{attribute 'qualified_only'}
{attribute 'strict'}
TYPE ERetargetType :
(
	not_retargeted := 0,
	primitive_target := 1,
	sequence_target := 2
);
END_TYPE

(* stored: Version 1.1.0.1, ProductVersion 3.1.4024.9
   DUT ERetargetType: Id {b4c5ac83-2993-4e71-8185-c38f70ce7ab7} *)
